Universal Robots PolyScope program: 5exIF.urp

Program 5exIF (installation=default directory=/home/ur/ursim-current/programs createdIn=5.11.8.1010444 lastSavedIn=5.11.8.1010444 robotSerialNumber=20195399999)
Calibrated DH parameters: a=[0, -0.24355, -0.2132, 0, 0, 0]; d=[0.15185, 0, 0, 0.13105, 0.08535, 0.0921]; alpha=[1.570796, 0, 0, 1.570796, -1.570796, 0]; deltaTheta=[0, 0, 0, 0, 0, 0]
BeforeStart
  Script file /home/ur/ursim-current/programs/Script/5_Ex_if.script
    | def If_Check(INPUT, digiIN):
    | 	if (digiIN == False):
    | 		if (get_standard_digital_out(INPUT) == True):
    | 			movel(p[0.10,-0.35,0.2,0.0,3.14,0.0], a=1, v=1)
    | 		end
    | 		if (get_standard_digital_out(INPUT) == False):
    | 			movel(p[-0.10,-0.35,0.4,0.0,3.14,0.0], a=1, v=1)
    | 		end
    | 	elif (digiIN == True):
    | 		if (get_standard_digital_in(INPUT) == True):
    | 			movel(p[0.0,-0.35,0.2,0.0,3.14,0.0], a=1, v=1)
    | 		end
    | 		if (get_standard_digital_in(INPUT) == False):
    | 			movel(p[0.0,-0.35,0.4,0.0,3.14,0.0], a=1, v=1)
    | 		end
    | 	end
    | end
  'Start position'
  x := 0.0
  y := -0.35
  z := 0.3
  rx := 0
  ry := 3.14
  rz := 0
  'going to start position via movej'
  Script: movej(p[x,y,z,rx,ry,rz],a=1,v=1)
Robot Program (runOnlyOnce=false)
  Wait Sleep waitTime=0.01
  Script: If_Check(0,False)
